// TIA Portal V20 export
TYPE "typeEm3Monitoring"
// stored: Access Published, Namespace Unit1
   STRUCT
      cmStatus { ExternalWritable := 'False'} : "Unit1.typeEm3MonitoringCmStatus";
      Jobstatus { S7_SetPoint := 'True'} : "Unit1.typeEm3MonitoringJobStatus";
      UserDefine { S7_SetPoint := 'True'} : "Unit1.typeEm3MonitoringUserDefine";
   END_STRUCT;
END_TYPE
